ABB RAPID module: Código RAPID

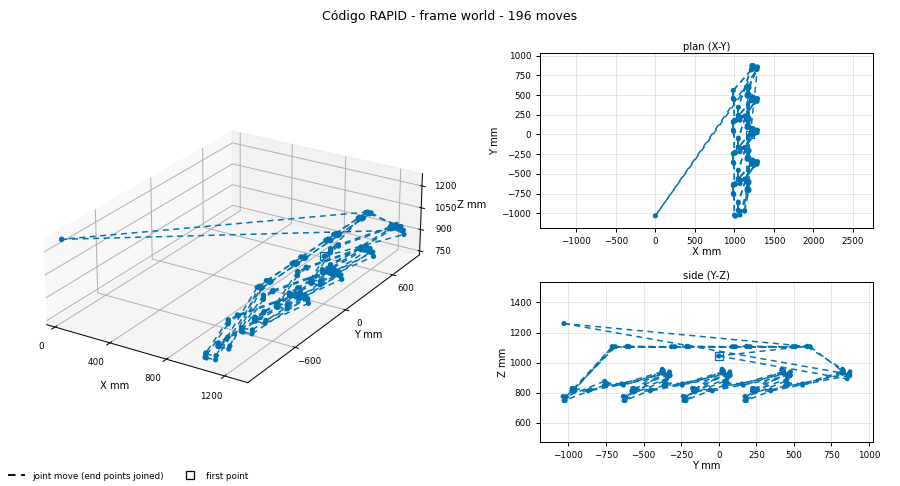
[picture p0: tool path of Código RAPID in frame world, 196 of 196 moves have a stored position in this frame; points joined in program order, loops and branches not executed]
MODULE Module1

    CONST robtarget HomeMesa:=[[1202.698927649,-0.006539298,1044.168012245],[0.707107406,0.00000178,0.707106156,-0.000001827],[-1,-1,0,1],[9E+09,9E+09,9E+09,0,0,0]];
    CONST robtarget Esperando:=[[0,-1030,1260],[0.500000347,0.500000347,0.499999653,-0.499999653],[-1,0,0,0],[9E+09,9E+09,9E+09,0,0,0]];
    CONST robtarget EsperandoMOVMesa:=[[-0.000045023,-1029.999947846,1260.000008248],[0.500000409,0.500000426,0.499999569,-0.499999596],[-2,0,0,0],[9E+09,9E+09,9E+09,180,0,0]];
    CONST robtarget HomeMesaDos:=[[1202.659544298,-0.000000047,1044.197481146],[0.706859937,0.00000059,0.707353539,0.00000059],[-1,-1,0,1],[9E+09,9E+09,9E+09,180,0,0]];
    CONST robtarget P1M1p1:=[[1294.65400628,854.62926339,891.446179617],[0.692157386,-0.14463472,0.692155179,-0.144638026],[0,0,-2,1],[9E+09,9E+09,9E+09,0,0,0]];
    CONST robtarget P1M1p2:=[[1240.529987934,870.337936268,911.143078471],[0.692157372,-0.144634704,0.692155207,-0.144637976],[0,0,-2,1],[9E+09,9E+09,9E+09,0,0,0]];
    CONST robtarget P1M1p3:=[[1227.787003999,873.332910408,915.014094682],[0.692157384,-0.144634674,0.692155202,-0.144637974],[0,0,-2,1],[9E+09,9E+09,9E+09,0,0,0]];
    CONST robtarget P1M1p4:=[[1222.239971547,870.997005167,915.013984808],[0.692157374,-0.144634683,0.692155208,-0.144637984],[0,0,-2,1],[9E+09,9E+09,9E+09,0,0,0]];
    CONST robtarget P1M1p5:=[[1050.485957284,345.048295942,811.300602855],[0.811802015,-0.047931337,0.525122518,0.250851384],[0,-1,0,1],[9E+09,9E+09,9E+09,0,0,0]];
    CONST robtarget P1M1p6:=[[1050.485947523,241.88479321,811.300594665],[0.811802009,-0.047931341,0.525122529,0.25085138],[0,-1,0,1],[9E+09,9E+09,9E+09,0,0,0]];
    CONST robtarget P1M1p7:=[[1057.883963041,232.826791757,811.30061261],[0.811802025,-0.047931351,0.525122498,0.250851392],[0,-1,0,1],[9E+09,9E+09,9E+09,0,0,0]];
    CONST robtarget P1M1p8:=[[1062.213995533,227.496594257,811.300605648],[0.81180201,-0.047931351,0.525122524,0.250851384],[0,-1,0,1],[9E+09,9E+09,9E+09,0,0,0]];
    CONST robtarget P1M1p9:=[[1069.026926797,223.929489315,811.300609594],[0.811802022,-0.047931351,0.525122506,0.250851385],[0,-1,0,1],[9E+09,9E+09,9E+09,0,0,0]];
    CONST robtarget P1M1p10:=[[1131.150947055,233.271896766,811.300583808],[0.811801999,-0.047931349,0.525122542,0.250851381],[0,-1,0,1],[9E+09,9E+09,9E+09,0,0,0]];
    CONST robtarget WaitMovMes1:=[[1202.698927649,-0.006539298,1044.168012245],[0.707107406,0.00000178,0.707106156,-0.000001827],[-1,-1,0,1],[9E+09,9E+09,9E+09,0,70,0]];
    CONST robtarget P1M1p11:=[[1185.930963599,608.173984403,1105.507035593],[0.707107406,0.000001819,0.707106156,-0.000001773],[0,0,-1,1],[9E+09,9E+09,9E+09,0,70,0]];
    CONST robtarget P1M1p12:=[[1185.930945833,510.993010056,1105.507039041],[0.707107406,0.000001805,0.707106157,-0.000001779],[0,0,-1,1],[9E+09,9E+09,9E+09,0,70,0]];
    CONST robtarget P1M2p1:=[[1287.081963914,823.391582063,930.460843736],[0.695385123,-0.126848673,0.695870584,-0.126937293],[0,0,-2,1],[9E+09,9E+09,9E+09,180,0,0]];
    CONST robtarget P1M2p2:=[[1232.892961405,829.555227251,930.460804282],[0.695385105,-0.126848727,0.69587059,-0.126937302],[0,0,-2,1],[9E+09,9E+09,9E+09,180,0,0]];
    CONST robtarget P1M2p3:=[[1217.609979435,827.253306759,930.460865831],[0.695385103,-0.12684871,0.695870597,-0.126937292],[0,0,-2,1],[9E+09,9E+09,9E+09,179.999964028,0,0]];
    CONST robtarget P1M2p4:=[[1214.009982986,817.991001642,930.460929766],[0.69538513,-0.126848699,0.695870573,-0.126937287],[0,0,-2,1],[9E+09,9E+09,9E+09,179.999964028,0,0]];
    CONST robtarget P1M2p5:=[[985.766137978,557.785104133,849.272525889],[0.8360719,0.017530565,0.547684306,0.026802208],[0,0,-1,1],[9E+09,9E+09,9E+09,179.999964028,0,0]];
    CONST robtarget P1M2p6:=[[985.766103061,457.716388895,849.272504479],[0.836071885,0.017530555,0.547684329,0.026802215],[0,0,-1,1],[9E+09,9E+09,9E+09,179.999964028,0,0]];
    CONST robtarget P1M2p7:=[[993.022666983,444.585787062,849.272520175],[0.836071898,0.017530568,0.547684309,0.026802211],[0,0,-1,1],[9E+09,9E+09,9E+09,179.999964028,0,0]];
    CONST robtarget P1M2p8:=[[1003.070938058,180.78768984,747.134418734],[0.807646496,0.209376596,0.514278881,0.19845859],[0,0,0,1],[9E+09,9E+09,9E+09,179.999964028,0,0]];
    CONST robtarget P1M2p9:=[[1013.977977246,173.442492628,747.1343984],[0.807646488,0.209376597,0.514278891,0.198458593],[0,0,0,1],[9E+09,9E+09,9E+09,179.999964028,0,0]];
    CONST robtarget P1M2p10:=[[1071.573952151,182.645606548,747.134407615],[0.807646513,0.209376602,0.514278845,0.198458605],[0,0,0,1],[9E+09,9E+09,9E+09,179.999964028,0,0]];
    CONST robtarget P1M2p11:=[[1185.930948842,588.452827755,1105.507011433],[0.707107409,0.000001805,0.707106154,-0.000001782],[0,0,-1,1],[9E+09,9E+09,9E+09,180,0,70]];
    CONST robtarget P1M2p12:=[[1185.93095036,492.129217368,1105.507026368],[0.707107404,0.000001839,0.707106158,-0.000001748],[0,0,-1,1],[9E+09,9E+09,9E+09,180,0,70]];
    CONST robtarget P2M1p1:=[[1294.653992166,454.43887346,891.446221022],[0.6921574,-0.144634673,0.692155181,-0.144638],[0,0,-1,1],[9E+09,9E+09,9E+09,0,0,0]];
    CONST robtarget P2M1p2:=[[1240.529984528,471.564123221,911.143162871],[0.692157397,-0.144634711,0.692155175,-0.144638006],[0,0,-1,1],[9E+09,9E+09,9E+09,0,0,0]];
    CONST robtarget P2M1p3:=[[1227.787003056,474.288594714,915.014113434],[0.69215739,-0.144634698,0.692155182,-0.144638018],[0,0,-1,1],[9E+09,9E+09,9E+09,0,0,0]];
    CONST robtarget P2M1p4:=[[1222.239953446,477.172888785,915.014065691],[0.692157397,-0.144634673,0.692155183,-0.144638],[0,0,-1,1],[9E+09,9E+09,9E+09,0,0,0]];
    CONST robtarget P2M1p5:=[[1050.485945509,-43.142440837,811.300594597],[0.811802019,-0.047931335,0.525122501,0.250851405],[-1,-1,0,1],[9E+09,9E+09,9E+09,0,0,0]];
    CONST robtarget P2M1p6:=[[1050.485952356,-156.521686759,811.300602341],[0.811802022,-0.047931365,0.525122503,0.250851385],[-1,-1,0,1],[9E+09,9E+09,9E+09,0,0,0]];
    CONST robtarget P2M1p7:=[[1057.883958265,-165.799494249,811.300583338],[0.811802006,-0.04793134,0.52512253,0.250851387],[-1,-1,0,1],[9E+09,9E+09,9E+09,0,0,0]];
    CONST robtarget P2M1p8:=[[1062.214006906,-168.868785565,811.300606455],[0.811802003,-0.047931336,0.525122535,0.250851386],[-1,-1,0,1],[9E+09,9E+09,9E+09,0,0,0]];
    CONST robtarget P2M1p9:=[[1069.026931582,-168.907600899,811.300592184],[0.811802005,-0.047931324,0.525122533,0.250851385],[-1,-1,0,1],[9E+09,9E+09,9E+09,0,0,0]];
    CONST robtarget P2M1p10:=[[1131.150939615,-165.021006485,811.300610263],[0.811802012,-0.047931365,0.525122515,0.250851394],[-1,-1,0,1],[9E+09,9E+09,9E+09,0,0,0]];
    CONST robtarget P2M1p11:=[[1185.930947732,209.275205026,1105.50703153],[0.707107405,0.00000183,0.707106157,-0.000001768],[0,0,-1,1],[9E+09,9E+09,9E+09,0,70,0]];
    CONST robtarget P2M1p12:=[[1185.930942037,104.027697243,1105.507044947],[0.707107412,0.000001825,0.70710615,-0.000001776],[0,0,-1,1],[9E+09,9E+09,9E+09,0,70,0]];
    CONST robtarget P3M1p1:=[[1294.653990055,54.307312118,891.446205655],[0.692157397,-0.144634698,0.692155177,-0.144638009],[0,0,-1,1],[9E+09,9E+09,9E+09,0,0,0]];
    CONST robtarget P3M1p2:=[[1240.529992729,70.522194984,911.143209882],[0.692157388,-0.144634701,0.692155185,-0.144638007],[0,0,-1,1],[9E+09,9E+09,9E+09,0,0,0]];
    CONST robtarget P3M1p3:=[[1227.787003035,75.815701326,915.01410237],[0.692157387,-0.144634691,0.692155191,-0.144637997],[0,0,-1,1],[9E+09,9E+09,9E+09,0,0,0]];
    CONST robtarget P3M1p4:=[[1222.239957402,75.077729076,915.014095799],[0.692157385,-0.144634702,0.692155189,-0.144638005],[0,0,-1,1],[9E+09,9E+09,9E+09,0,0,0]];
    CONST robtarget P3M1p5:=[[1050.485952963,-456.006186482,811.300606987],[0.811802017,-0.047931347,0.525122507,0.250851398],[-1,-1,0,1],[9E+09,9E+09,9E+09,0,0,0]];
    CONST robtarget P3M1p6:=[[1050.485949852,-556.041703529,811.300612034],[0.811802017,-0.047931384,0.525122509,0.250851386],[-1,-1,0,1],[9E+09,9E+09,9E+09,0,0,0]];
    CONST robtarget P3M1p7:=[[1057.883966107,-571.807786887,811.300587052],[0.811802004,-0.047931339,0.525122524,0.250851405],[-1,-1,0,1],[9E+09,9E+09,9E+09,0,0,0]];
    CONST robtarget P3M1p8:=[[1062.214003211,-570.695858455,811.30060674],[0.811802022,-0.047931361,0.525122502,0.25085139],[-1,-1,0,1],[9E+09,9E+09,9E+09,0,0,0]];
    CONST robtarget P3M1p9:=[[1069.02692125,-578.673501326,811.300606016],[0.811802025,-0.047931285,0.525122514,0.250851369],[-1,-1,0,1],[9E+09,9E+09,9E+09,0,0,0]];
    CONST robtarget P3M1p10:=[[1131.150956875,-570.701987213,811.300598508],[0.811802018,-0.047931365,0.525122499,0.250851406],[-1,-1,0,1],[9E+09,9E+09,9E+09,0,0,0]];
    CONST robtarget P3M1p11:=[[1185.930947007,-197.514283951,1105.507037733],[0.707107409,0.000001821,0.707106153,-0.00000177],[-1,-1,0,1],[9E+09,9E+09,9E+09,0,70,0]];
    CONST robtarget P3M1p12:=[[1185.930941597,-293.197607054,1105.507038781],[0.70710741,0.000001841,0.707106152,-0.000001751],[-1,-1,0,1],[9E+09,9E+09,9E+09,0,70,0]];
    CONST robtarget P4M1p1:=[[1294.653989986,-345.662907333,891.446190924],[0.692157389,-0.144634676,0.69215519,-0.144638004],[-1,-1,0,1],[9E+09,9E+09,9E+09,0,0,0]];
    CONST robtarget P4M1p2:=[[1240.530000685,-329.603196599,911.143191009],[0.692157385,-0.1446347,0.692155189,-0.144638003],[-1,-1,0,1],[9E+09,9E+09,9E+09,0,0,0]];
    CONST robtarget P4M1p3:=[[1227.787004205,-322.940201758,915.014096584],[0.692157384,-0.144634687,0.692155193,-0.144638003],[-1,-1,0,1],[9E+09,9E+09,9E+09,0,0,0]];
    CONST robtarget P4M1p4:=[[1222.23995583,-327.607308393,915.014097519],[0.692157385,-0.144634701,0.692155189,-0.144638006],[-1,-1,0,1],[9E+09,9E+09,9E+09,0,0,0]];
    CONST robtarget P4M1p5:=[[1050.485949411,-869.115712575,811.300612218],[0.811802019,-0.047931325,0.525122516,0.250851378],[-1,-1,0,1],[9E+09,9E+09,9E+09,0,0,0]];
    CONST robtarget P4M1p6:=[[1050.485974835,-958.232069962,811.300585733],[0.811802011,-0.047931384,0.525122503,0.250851418],[-1,-1,0,1],[9E+09,9E+09,9E+09,0,0,0]];
    CONST robtarget P4M1p7:=[[1057.88399001,-975.404649155,811.30060734],[0.811802006,-0.047931318,0.525122528,0.250851396],[-1,-1,0,1],[9E+09,9E+09,9E+09,0,0,0]];
    CONST robtarget P4M1p8:=[[1062.214034381,-973.918880257,811.300571248],[0.811802021,-0.047931344,0.525122509,0.250851381],[-1,-1,0,1],[9E+09,9E+09,9E+09,0,0,0]];
    CONST robtarget P4M1p9:=[[1069.026916149,-978.501930546,811.300562057],[0.811802023,-0.047931276,0.525122506,0.250851395],[-1,-1,0,1],[9E+09,9E+09,9E+09,0,0,0]];
    CONST robtarget P4M1p10:=[[1131.150931317,-972.859035446,811.300552906],[0.811802013,-0.047931366,0.525122516,0.250851386],[-1,-1,0,1],[9E+09,9E+09,9E+09,0,0,0]];
    CONST robtarget P4M1p11:=[[1185.930958357,-596.032669183,1105.507027322],[0.70710741,0.000001831,0.707106152,-0.000001743],[-1,-1,0,1],[9E+09,9E+09,9E+09,0,70,0]];
    CONST robtarget P4M1p12:=[[1185.930974143,-694.807857486,1105.507021321],[0.707107404,0.000001822,0.707106159,-0.000001766],[-1,-1,0,1],[9E+09,9E+09,9E+09,0,70,0]];
    CONST robtarget TurnMesa:=[[1202.698927649,-0.006539298,1044.168012245],[0.707107406,0.00000178,0.707106156,-0.000001827],[-1,-1,0,1],[9E+09,9E+09,9E+09,0,180,0]];
    CONST robtarget P5M1p1:=[[1287.51280176,856.97594778,918.184846829],[0.692157388,-0.144634706,0.692155182,-0.144638018],[0,0,-2,1],[9E+09,9E+09,9E+09,0,180,0]];
    CONST robtarget P5M1p2:=[[1240.529986137,870.338041259,927.422439494],[0.69215738,-0.144634719,0.692155189,-0.144638011],[0,0,-2,1],[9E+09,9E+09,9E+09,0,180,0]];
    CONST robtarget P5M1p3:=[[1227.787003999,873.332910408,938.961164099],[0.692157384,-0.144634674,0.692155202,-0.144637974],[0,0,-2,1],[9E+09,9E+09,9E+09,0,180,0]];
    CONST robtarget P5M1p4:=[[1222.239971547,870.997005167,929.420285517],[0.692157374,-0.144634683,0.692155208,-0.144637984],[0,0,-2,1],[9E+09,9E+09,9E+09,0,180,0]];
    CONST robtarget P5M1p5:=[[1050.485957284,345.048295942,818.663201985],[0.811802015,-0.047931337,0.525122518,0.250851384],[0,-1,0,1],[9E+09,9E+09,9E+09,0,180,0]];
    CONST robtarget P5M1p6:=[[1050.485947523,241.88479321,824.353888262],[0.811802009,-0.047931341,0.525122529,0.25085138],[0,-1,0,1],[9E+09,9E+09,9E+09,0,180,0]];
    CONST robtarget P5M1p7:=[[1057.883963041,232.826791757,825.451999614],[0.811802025,-0.047931351,0.525122498,0.250851392],[0,-1,0,1],[9E+09,9E+09,9E+09,0,180,0]];
    CONST robtarget P5M1p8:=[[1062.213995533,227.496594257,827.795822741],[0.81180201,-0.047931351,0.525122524,0.250851384],[0,-1,0,1],[9E+09,9E+09,9E+09,0,180,0]];
    CONST robtarget P5M1p9:=[[1069.026926797,223.929489315,828.586291332],[0.811802022,-0.047931351,0.525122506,0.250851385],[0,-1,0,1],[9E+09,9E+09,9E+09,0,180,0]];
    CONST robtarget P5M1p10:=[[1131.150947055,233.271896766,826.446924128],[0.811801999,-0.047931349,0.525122542,0.250851381],[0,-1,0,1],[9E+09,9E+09,9E+09,0,180,0]];
    CONST robtarget P5M1p11:=[[1160.941867257,608.173984403,1105.507035593],[0.707107406,0.000001819,0.707106156,-0.000001773],[0,0,-1,1],[9E+09,9E+09,9E+09,0,250,0]];
    CONST robtarget P5M1p12:=[[1160.941943935,507.930686372,1105.50702957],[0.707107404,0.000001805,0.707106158,-0.000001799],[0,0,-1,1],[9E+09,9E+09,9E+09,0,250,0]];
    CONST robtarget P6M1p1:=[[1287.512992537,455.226798507,918.184930623],[0.692157396,-0.14463471,0.692155172,-0.144638022],[0,0,-1,1],[9E+09,9E+09,9E+09,0,180,0]];
    CONST robtarget P6M1p2:=[[1240.530007914,466.532478263,927.422537461],[0.692157392,-0.14463468,0.692155189,-0.144637993],[0,0,-1,1],[9E+09,9E+09,9E+09,0,180,0]];
    CONST robtarget P6M1p3:=[[1227.787004184,477.674601054,938.961099959],[0.692157386,-0.144634703,0.692155187,-0.14463801],[0,0,-1,1],[9E+09,9E+09,9E+09,0,180,0]];
    CONST robtarget P6M1p4:=[[1222.239961288,469.693192082,929.420433939],[0.69215739,-0.144634696,0.692155187,-0.144637993],[0,0,-1,1],[9E+09,9E+09,9E+09,0,180,0]];
    CONST robtarget P6M1p5:=[[1050.485946451,-57.179143328,818.663195557],[0.81180201,-0.04793132,0.525122533,0.250851372],[-1,-1,0,1],[9E+09,9E+09,9E+09,0,180,0]];
    CONST robtarget P6M1p6:=[[1050.485945699,-158.82959493,824.353885396],[0.811802018,-0.047931342,0.525122505,0.250851399],[-1,-1,0,1],[9E+09,9E+09,9E+09,0,180,0]];
    CONST robtarget P6M1p7:=[[1057.883963528,-170.135898305,825.452052847],[0.811802002,-0.047931347,0.525122534,0.250851389],[-1,-1,0,1],[9E+09,9E+09,9E+09,0,180,0]];
    CONST robtarget P6M1p8:=[[1062.213999596,-173.347293692,827.795942722],[0.811802007,-0.047931318,0.525122528,0.250851393],[-1,-1,0,1],[9E+09,9E+09,9E+09,0,180,0]];
    CONST robtarget P6M1p9:=[[1069.02693064,-173.705298015,828.586300968],[0.811802009,-0.047931353,0.525122532,0.250851372],[-1,-1,0,1],[9E+09,9E+09,9E+09,0,180,0]];
    CONST robtarget P6M1p10:=[[1131.15094581,-164.207103159,826.447012387],[0.811802001,-0.047931347,0.525122543,0.250851374],[-1,-1,0,1],[9E+09,9E+09,9E+09,0,180,0]];
    CONST robtarget P7M1p1:=[[1287.5130039,55.947838621,918.184889325],[0.69215739,-0.1446347,0.692155182,-0.14463801],[0,0,-1,1],[9E+09,9E+09,9E+09,0,180,0]];
    CONST robtarget P7M1p2:=[[1240.529993957,74.049824175,927.422605126],[0.692157388,-0.144634689,0.69215519,-0.144637995],[0,0,-1,1],[9E+09,9E+09,9E+09,0,180,0]];
    CONST robtarget P7M1p3:=[[1227.786997792,73.453377394,938.961112671],[0.692157392,-0.144634702,0.69215518,-0.144638014],[0,0,-1,1],[9E+09,9E+09,9E+09,0,180,0]];
    CONST robtarget P7M1p4:=[[1222.239945235,71.066640414,929.420450662],[0.692157398,-0.144634691,0.692155178,-0.144638003],[0,0,-1,1],[9E+09,9E+09,9E+09,0,180,0]];
    CONST robtarget P7M1p5:=[[1050.485943723,-450.547007586,818.663211154],[0.811802031,-0.047931305,0.525122495,0.250851388],[-1,-1,0,1],[9E+09,9E+09,9E+09,0,180,0]];
    CONST robtarget P7M1p6:=[[1050.485951308,-555.654089777,824.353906332],[0.811802023,-0.047931345,0.525122502,0.25085139],[-1,-1,0,1],[9E+09,9E+09,9E+09,0,180,0]];
    CONST robtarget P7M1p7:=[[1057.883971379,-565.529692139,825.452046896],[0.811802007,-0.047931352,0.525122531,0.250851378],[-1,-1,0,1],[9E+09,9E+09,9E+09,0,180,0]];
    CONST robtarget P7M1p8:=[[1062.214013779,-572.186553681,827.795959878],[0.811802015,-0.047931347,0.525122524,0.250851369],[-1,-1,0,1],[9E+09,9E+09,9E+09,0,180,0]];
    CONST robtarget P7M1p9:=[[1069.026937537,-571.189267924,828.58630883],[0.811802019,-0.047931339,0.525122522,0.250851362],[-1,-1,0,1],[9E+09,9E+09,9E+09,0,180,0]];
    CONST robtarget P7M1p10:=[[1131.150959132,-562.660960026,826.447030815],[0.81180201,-0.047931389,0.525122518,0.25085139],[-1,-1,0,1],[9E+09,9E+09,9E+09,0,180,0]];
    CONST robtarget P6M1p11:=[[1160.941935741,207.369302139,1105.50703556],[0.707107406,0.000001794,0.707106157,-0.00000179],[0,0,-1,1],[9E+09,9E+09,9E+09,0,250,0]];
    CONST robtarget P6M1p12:=[[1160.941940446,113.055695188,1105.507031057],[0.707107406,0.00000181,0.707106156,-0.000001778],[0,0,-1,1],[9E+09,9E+09,9E+09,0,250,0]];
    CONST robtarget P7M1p11:=[[1160.941939753,-202.48499324,1105.507031431],[0.707107406,0.00000177,0.707106157,-0.000001802],[-1,-1,0,1],[9E+09,9E+09,9E+09,0,250,0]];
    CONST robtarget P7M1p12:=[[1160.941939671,-291.239289206,1105.507030754],[0.70710741,0.000001779,0.707106153,-0.000001789],[-1,-1,0,1],[9E+09,9E+09,9E+09,0,250,0]];
    CONST robtarget P8M1p1:=[[1287.513001746,-341.869412046,918.184887932],[0.692157384,-0.144634701,0.69215519,-0.144638003],[-1,-1,0,1],[9E+09,9E+09,9E+09,0,180,0]];
    CONST robtarget P8M1p2:=[[1240.529989369,-331.61750501,927.422616777],[0.692157392,-0.144634697,0.692155182,-0.144638007],[-1,-1,0,1],[9E+09,9E+09,9E+09,0,180,0]];
    CONST robtarget P8M1p3:=[[1227.787006733,-328.052388339,938.961097781],[0.692157382,-0.144634706,0.692155192,-0.144638003],[-1,-1,0,1],[9E+09,9E+09,9E+09,0,180,0]];
    CONST robtarget P8M1p4:=[[1222.23995944,-330.109669308,929.420486052],[0.692157392,-0.144634689,0.692155187,-0.144637993],[-1,-1,0,1],[9E+09,9E+09,9E+09,0,180,0]];
    CONST robtarget P8M1p5:=[[1050.485978825,-853.276272126,818.663203151],[0.81180201,-0.047931328,0.525122523,0.250851391],[-1,-1,0,1],[9E+09,9E+09,9E+09,0,180,0]];
    CONST robtarget P8M1p6:=[[1050.485957025,-958.593434584,824.353874621],[0.811802012,-0.047931339,0.525122527,0.250851375],[-1,-1,0,1],[9E+09,9E+09,9E+09,0,180,0]];
    CONST robtarget P8M1p7:=[[1057.883978797,-972.736439335,825.452068596],[0.811802005,-0.047931352,0.525122524,0.250851402],[-1,-1,0,1],[9E+09,9E+09,9E+09,0,180,0]];
    CONST robtarget P8M1p8:=[[1062.214032655,-971.575289729,827.795997264],[0.811802013,-0.047931351,0.525122523,0.250851377],[-1,-1,0,1],[9E+09,9E+09,9E+09,0,180,0]];
    CONST robtarget P8M1p9:=[[1069.026937278,-976.446817795,828.586268385],[0.811802017,-0.047931332,0.525122513,0.250851388],[-1,-1,0,1],[9E+09,9E+09,9E+09,0,180,0]];
    CONST robtarget P8M1p10:=[[1131.150976145,-960.905988949,826.447126012],[0.811802005,-0.047931424,0.525122525,0.250851386],[-1,-1,0,1],[9E+09,9E+09,9E+09,0,180,0]];
    CONST robtarget P8M1p11:=[[1160.941952888,-598.731774088,1105.507053568],[0.707107405,0.000001738,0.707106157,-0.000001833],[-1,-1,0,1],[9E+09,9E+09,9E+09,0,250,0]];
    CONST robtarget P8M1p12:=[[1160.941938987,-686.786158028,1105.507050864],[0.70710742,0.00000173,0.707106142,-0.00000184],[-1,-1,0,1],[9E+09,9E+09,9E+09,0,250,0]];
    CONST robtarget P2M2p1:=[[1287.081942915,423.299490757,930.460887717],[0.695385109,-0.1268487,0.695870591,-0.126937301],[0,0,-1,1],[9E+09,9E+09,9E+09,180,0,0]];
    CONST robtarget P2M2p2:=[[1232.892982774,430.194982931,930.460817958],[0.695385103,-0.126848709,0.695870593,-0.126937314],[0,0,-1,1],[9E+09,9E+09,9E+09,180,0,0]];
    CONST robtarget P2M2p3:=[[1217.609985933,434.601968819,930.460907436],[0.695385116,-0.126848706,0.69587058,-0.126937316],[0,0,-1,1],[9E+09,9E+09,9E+09,180,0,0]];
    CONST robtarget P2M2p4:=[[1214.009978094,428.335193568,930.460893887],[0.695385201,-0.126848703,0.6958705,-0.126937292],[0,0,-1,1],[9E+09,9E+09,9E+09,180,0,0]];
    CONST robtarget P2M2p5:=[[985.766084152,163.956301034,849.272497669],[0.836071892,0.017530565,0.547684317,0.02680222],[0,0,-1,1],[9E+09,9E+09,9E+09,180,0,0]];
    CONST robtarget P2M2p6:=[[985.7660988,48.871628128,849.272538428],[0.836071912,0.01753054,0.547684287,0.02680222],[0,0,0,1],[9E+09,9E+09,9E+09,180,0,0]];
    CONST robtarget P2M2p7:=[[993.022664863,36.972499936,849.272528775],[0.8360719,0.017530569,0.547684306,0.02680221],[0,0,0,1],[9E+09,9E+09,9E+09,180,0,0]];
    CONST robtarget P2M2p8:=[[1003.0709257,-228.723692996,747.134400051],[0.807646484,0.209376611,0.514278887,0.198458605],[-1,-1,0,1],[9E+09,9E+09,9E+09,180,0,0]];
    CONST robtarget P2M2p9:=[[1013.977992175,-232.129697703,747.134426921],[0.807646515,0.209376583,0.514278857,0.198458586],[-1,-1,0,1],[9E+09,9E+09,9E+09,180,0,0]];
    CONST robtarget P2M2p10:=[[1071.573958877,-217.594289105,747.13441737],[0.80764653,0.209376599,0.514278819,0.198458606],[-1,-1,0,1],[9E+09,9E+09,9E+09,180,0,0]];
    CONST robtarget P2M2p11:=[[1185.930950239,187.675889547,1105.507032353],[0.707107407,0.000001823,0.707106155,-0.000001789],[0,0,-1,1],[9E+09,9E+09,9E+09,180,0,70]];
    CONST robtarget P2M2p12:=[[1185.930943233,95.529018748,1105.507041573],[0.70710741,0.000001834,0.707106153,-0.000001752],[0,0,-1,1],[9E+09,9E+09,9E+09,180,0,70]];
    CONST robtarget P3M2p1:=[[1287.081941566,21.413279151,930.460887197],[0.695385111,-0.126848701,0.695870588,-0.126937304],[0,0,-1,1],[9E+09,9E+09,9E+09,180,0,0]];
    CONST robtarget P3M2p2:=[[1232.892967953,28.987158369,930.460840817],[0.695385113,-0.126848699,0.695870587,-0.126937303],[0,0,-1,1],[9E+09,9E+09,9E+09,180,0,0]];
    CONST robtarget P3M2p3:=[[1217.60998262,34.410408763,930.460892089],[0.695385108,-0.126848696,0.695870593,-0.126937298],[0,0,-1,1],[9E+09,9E+09,9E+09,180,0,0]];
    CONST robtarget P3M2p4:=[[1214.009984068,31.687269665,930.460885715],[0.695385201,-0.126848699,0.695870499,-0.126937302],[0,0,-1,1],[9E+09,9E+09,9E+09,180,0,0]];
    CONST robtarget P3M2p5:=[[985.766085968,-242.896799387,849.27250766],[0.836071903,0.017530563,0.547684302,0.026802208],[-1,-1,0,1],[9E+09,9E+09,9E+09,180,0,0]];
    CONST robtarget P3M2p6:=[[985.766092573,-352.969410753,849.272514142],[0.836071905,0.017530541,0.547684299,0.026802214],[-1,-1,0,1],[9E+09,9E+09,9E+09,180,0,0]];
    CONST robtarget P3M2p7:=[[993.022662409,-364.919381115,849.272509954],[0.83607191,0.017530563,0.547684291,0.026802221],[-1,-1,0,1],[9E+09,9E+09,9E+09,180,0,0]];
    CONST robtarget P3M2p8:=[[1003.070932407,-628.513700129,747.134415648],[0.807646507,0.209376596,0.51427886,0.198458599],[-1,-1,0,1],[9E+09,9E+09,9E+09,180,0,0]];
    CONST robtarget P3M2p9:=[[1013.977996648,-630.345557467,747.134426277],[0.807646526,0.209376596,0.514278831,0.198458594],[-1,-1,0,1],[9E+09,9E+09,9E+09,180,0,0]];
    CONST robtarget P3M2p10:=[[1071.573965127,-622.825071858,747.134417066],[0.807646527,0.209376586,0.514278841,0.198458579],[-1,-1,0,1],[9E+09,9E+09,9E+09,180,0,0]];
    CONST robtarget P3M2p11:=[[1185.930946533,-213.064594931,1105.507036914],[0.707107409,0.000001806,0.707106153,-0.000001799],[-1,-1,0,1],[9E+09,9E+09,9E+09,180,0,70]];
    CONST robtarget P3M2p12:=[[1185.930948227,-314.722485056,1105.507040307],[0.707107408,0.0000018,0.707106154,-0.000001796],[-1,-1,0,1],[9E+09,9E+09,9E+09,180,0,70]];
    CONST robtarget P4M2p1:=[[1287.081937875,-376.65299891,930.46088109],[0.695385101,-0.126848707,0.695870596,-0.126937313],[-1,-1,0,1],[9E+09,9E+09,9E+09,180,0,0]];
    CONST robtarget P4M2p2:=[[1232.892982402,-370.043883982,930.460878188],[0.695385103,-0.126848708,0.695870596,-0.126937299],[-1,-1,0,1],[9E+09,9E+09,9E+09,180,0,0]];
    CONST robtarget P4M2p3:=[[1217.609984921,-367.718324415,930.460875748],[0.695385104,-0.126848682,0.695870599,-0.126937299],[-1,-1,0,1],[9E+09,9E+09,9E+09,180,0,0]];
    CONST robtarget P4M2p4:=[[1214.009976161,-372.318596656,930.460900471],[0.695385203,-0.126848704,0.695870495,-0.126937304],[-1,-1,0,1],[9E+09,9E+09,9E+09,180,0,0]];
    CONST robtarget P4M2p5:=[[985.766087685,-634.35829981,849.272500138],[0.836071901,0.017530576,0.547684304,0.02680221],[-1,-1,0,1],[9E+09,9E+09,9E+09,180,0,0]];
    CONST robtarget P4M2p6:=[[985.766074892,-747.923087794,849.272525035],[0.836071911,0.017530544,0.54768429,0.026802203],[-1,-1,0,1],[9E+09,9E+09,9E+09,180,0,0]];
    CONST robtarget P4M2p7:=[[993.022657334,-761.317316304,849.272520024],[0.836071894,0.017530573,0.547684315,0.026802205],[-1,-1,0,1],[9E+09,9E+09,9E+09,180,0,0]];
    CONST robtarget P4M2p8:=[[1003.070923563,-1027.52495413,747.134373101],[0.807646499,0.209376593,0.514278873,0.198458599],[-1,-1,0,1],[9E+09,9E+09,9E+09,180,0,0]];
    CONST robtarget P4M2p9:=[[1013.978011173,-1030.027003938,747.13443015],[0.807646524,0.209376598,0.514278843,0.19845857],[-1,-1,0,1],[9E+09,9E+09,9E+09,180,0,0]];
    CONST robtarget P4M2p10:=[[1071.573975734,-1021.038991656,747.134380172],[0.807646517,0.209376617,0.514278826,0.198458622],[-1,-1,0,1],[9E+09,9E+09,9E+09,180,0,0]];
    CONST robtarget P4M2p11:=[[1185.930951631,-611.718126779,1105.50700953],[0.707107393,0.000001797,0.707106169,-0.000001819],[-1,-1,0,1],[9E+09,9E+09,9E+09,180,0,70]];
    CONST robtarget P4M2p12:=[[1185.930932946,-710.183230163,1105.507022383],[0.707107409,0.000001848,0.707106153,-0.000001799],[-1,-1,0,1],[9E+09,9E+09,9E+09,180,0,70]];
    CONST robtarget P5M2p1:=[[1287.081963937,823.39158063,956.573530849],[0.695385109,-0.126848705,0.695870584,-0.126937335],[0,0,-2,1],[9E+09,9E+09,9E+09,180,0,180]];
    CONST robtarget P5M2p2:=[[1232.892961405,829.555227251,946.574452649],[0.695385105,-0.126848727,0.69587059,-0.126937302],[0,0,-2,1],[9E+09,9E+09,9E+09,180,0,180]];
    CONST robtarget P5M2p3:=[[1217.609979435,827.253306759,946.518852379],[0.695385103,-0.12684871,0.695870597,-0.126937292],[0,0,-2,1],[9E+09,9E+09,9E+09,180,0,180]];
    CONST robtarget P5M2p4:=[[1214.009981629,817.991000196,938.720837099],[0.695385178,-0.126848677,0.695870529,-0.126937286],[0,0,-2,1],[9E+09,9E+09,9E+09,180,0,180]];
    CONST robtarget P5M2p5:=[[985.766096585,557.785078701,859.297655027],[0.836071893,0.017530567,0.547684317,0.026802216],[0,0,-1,1],[9E+09,9E+09,9E+09,180,0,180]];
    CONST robtarget P5M2p6:=[[985.766102672,457.71639088,863.722348668],[0.836071888,0.017530541,0.547684325,0.026802215],[0,0,-1,1],[9E+09,9E+09,9E+09,180,0,180]];
    CONST robtarget P5M2p7:=[[993.022666983,444.585787062,876.038087888],[0.836071898,0.017530568,0.547684309,0.026802211],[0,0,-1,1],[9E+09,9E+09,9E+09,180,0,180]];
    CONST robtarget P5M2p8:=[[1003.070938058,180.78768984,772.485475081],[0.807646496,0.209376596,0.514278881,0.19845859],[0,0,0,1],[9E+09,9E+09,9E+09,180,0,180]];
    CONST robtarget P5M2p9:=[[1013.977977246,173.442492628,774.873565047],[0.807646488,0.209376597,0.514278891,0.198458593],[0,0,0,1],[9E+09,9E+09,9E+09,180,0,180]];
    CONST robtarget P5M2p10:=[[1071.573952151,182.645606548,771.890741042],[0.807646513,0.209376602,0.514278845,0.198458605],[0,0,0,1],[9E+09,9E+09,9E+09,180,0,180]];
    CONST robtarget P5M2p11:=[[1159.718533142,588.452792411,1109.600135223],[0.707107409,0.000001816,0.707106154,-0.000001793],[0,0,-1,1],[9E+09,9E+09,9E+09,180,0,250]];
    CONST robtarget P5M2p12:=[[1158.995416353,492.129217368,1105.507026368],[0.707107404,0.000001839,0.707106158,-0.000001748],[0,0,-1,1],[9E+09,9E+09,9E+09,180,0,250]];
    CONST robtarget P6M2p1:=[[1287.081942874,420.03000634,956.573432269],[0.69538511,-0.126848716,0.695870585,-0.126937314],[0,0,-1,1],[9E+09,9E+09,9E+09,180,0,180]];
    CONST robtarget P6M2p2:=[[1232.892962329,427.246392285,946.574422328],[0.695385114,-0.126848699,0.695870586,-0.1269373],[0,0,-1,1],[9E+09,9E+09,9E+09,180,0,180]];
    CONST robtarget P6M2p3:=[[1217.609978669,431.701906072,946.518805799],[0.695385111,-0.126848707,0.695870589,-0.126937293],[0,0,-1,1],[9E+09,9E+09,9E+09,180,0,180]];
    CONST robtarget P6M2p4:=[[1214.009982742,425.527880519,938.720915064],[0.695385203,-0.12684869,0.6958705,-0.126937297],[0,0,-1,1],[9E+09,9E+09,9E+09,180,0,180]];
    CONST robtarget P6M2p5:=[[985.766086342,153.560690225,859.297582324],[0.836071893,0.01753055,0.547684317,0.026802227],[0,0,-1,1],[9E+09,9E+09,9E+09,180,0,180]];
    CONST robtarget P6M2p6:=[[985.766094733,57.430100166,863.7224247],[0.83607191,0.01753054,0.54768429,0.026802231],[0,0,-1,1],[9E+09,9E+09,9E+09,180,0,180]];
    CONST robtarget P6M2p7:=[[993.022659885,38.244880974,876.038102784],[0.836071901,0.01753056,0.547684304,0.02680221],[0,0,0,1],[9E+09,9E+09,9E+09,180,0,180]];
    CONST robtarget P6M2p8:=[[1003.070925748,-229.263088707,772.48562708],[0.807646486,0.20937661,0.514278885,0.198458604],[-1,-1,0,1],[9E+09,9E+09,9E+09,180,0,180]];
    CONST robtarget P6M2p9:=[[1013.977986109,-237.325696282,774.87363237],[0.807646493,0.209376602,0.514278882,0.19845859],[-1,-1,0,1],[9E+09,9E+09,9E+09,180,0,180]];
    CONST robtarget P6M2p10:=[[1071.5739537,-217.291392288,771.890844811],[0.807646529,0.209376602,0.514278817,0.198458612],[-1,-1,0,1],[9E+09,9E+09,9E+09,180,0,180]];
    CONST robtarget P6M2p11:=[[1159.718967768,185.056293345,1109.599968508],[0.707107406,0.000001782,0.707106157,-0.000001809],[0,0,-1,1],[9E+09,9E+09,9E+09,180,0,250]];
    CONST robtarget P6M2p12:=[[1158.995007718,88.334741652,1105.507040855],[0.707107407,0.000001845,0.707106155,-0.000001754],[0,0,-1,1],[9E+09,9E+09,9E+09,180,0,250]];
    CONST robtarget P7M2p1:=[[1287.081938268,21.890938974,956.57351039],[0.695385113,-0.126848703,0.695870585,-0.126937308],[0,0,-1,1],[9E+09,9E+09,9E+09,180,0,180]];
    CONST robtarget P7M2p2:=[[1232.89296877,24.144487835,946.574415906],[0.695385111,-0.126848702,0.695870587,-0.126937306],[0,0,-1,1],[9E+09,9E+09,9E+09,180,0,180]];
    CONST robtarget P7M2p3:=[[1217.609978031,30.830878938,946.518813687],[0.695385117,-0.126848694,0.695870584,-0.126937301],[0,0,-1,1],[9E+09,9E+09,9E+09,180,0,180]];
    CONST robtarget P7M2p4:=[[1214.009982564,27.014900378,938.720897759],[0.695385201,-0.126848692,0.695870501,-0.126937294],[0,0,-1,1],[9E+09,9E+09,9E+09,180,0,180]];
    CONST robtarget P7M2p5:=[[985.766097151,-242.694294826,859.297602362],[0.836071894,0.017530542,0.547684315,0.026802225],[-1,-1,0,1],[9E+09,9E+09,9E+09,180,0,180]];
    CONST robtarget P7M2p6:=[[985.766099125,-352.829883584,863.722418914],[0.836071911,0.017530532,0.547684288,0.026802244],[-1,-1,0,1],[9E+09,9E+09,9E+09,180,0,180]];
    CONST robtarget P7M2p7:=[[993.022660819,-362.965703245,876.038079243],[0.836071881,0.017530584,0.547684334,0.026802208],[-1,-1,0,1],[9E+09,9E+09,9E+09,180,0,180]];
    CONST robtarget P7M2p8:=[[1003.070948251,-628.753993071,772.485658081],[0.807646515,0.209376563,0.514278862,0.198458594],[-1,-1,0,1],[9E+09,9E+09,9E+09,180,0,180]];
    CONST robtarget P7M2p9:=[[1013.977972406,-636.678405216,774.873711553],[0.807646507,0.209376587,0.514278867,0.19845859],[-1,-1,0,1],[9E+09,9E+09,9E+09,180,0,180]];
    CONST robtarget P7M2p10:=[[1071.573961903,-618.428809445,771.890835972],[0.80764652,0.209376611,0.514278821,0.198458631],[-1,-1,0,1],[9E+09,9E+09,9E+09,180,0,180]];
    CONST robtarget P7M2p11:=[[1159.718972896,-211.532582055,1109.599963477],[0.707107406,0.000001788,0.707106156,-0.000001804],[-1,-1,0,1],[9E+09,9E+09,9E+09,180,0,250]];
    CONST robtarget P7M2p12:=[[1158.995014498,-312.213370951,1105.507037983],[0.707107405,0.000001806,0.707106158,-0.000001779],[-1,-1,0,1],[9E+09,9E+09,9E+09,180,0,250]];
    CONST robtarget P8M2p1:=[[1287.081946207,-375.923966976,956.573509614],[0.695385119,-0.126848699,0.695870583,-0.126937291],[-1,-1,0,1],[9E+09,9E+09,9E+09,180,0,180]];
    CONST robtarget P8M2p2:=[[1232.892963196,-371.870194113,946.57442583],[0.69538511,-0.1268487,0.695870588,-0.126937308],[-1,-1,0,1],[9E+09,9E+09,9E+09,180,0,180]];
    CONST robtarget P8M2p3:=[[1217.609976063,-368.396995577,946.518812071],[0.695385112,-0.126848691,0.695870589,-0.126937305],[-1,-1,0,1],[9E+09,9E+09,9E+09,180,0,180]];
    CONST robtarget P8M2p4:=[[1214.009980014,-377.44629786,938.720900615],[0.695385192,-0.126848698,0.695870507,-0.126937304],[-1,-1,0,1],[9E+09,9E+09,9E+09,180,0,180]];
    CONST robtarget P8M2p5:=[[985.766102139,-645.865947475,859.297609634],[0.83607191,0.017530516,0.54768429,0.026802252],[-1,-1,0,1],[9E+09,9E+09,9E+09,180,0,180]];
    CONST robtarget P8M2p6:=[[985.766111508,-745.745453353,863.722406721],[0.836071896,0.017530535,0.547684312,0.026802244],[-1,-1,0,1],[9E+09,9E+09,9E+09,180,0,180]];
    CONST robtarget P8M2p7:=[[993.022651473,-759.598032516,876.03808882],[0.836071897,0.017530614,0.547684309,0.026802201],[-1,-1,0,1],[9E+09,9E+09,9E+09,180,0,180]];
    CONST robtarget P8M2p8:=[[1003.070942622,-1018.707021048,772.485722249],[0.807646501,0.209376576,0.514278888,0.198458571],[-1,-1,0,1],[9E+09,9E+09,9E+09,180,0,180]];
    CONST robtarget P8M2p9:=[[1013.978003834,-1036.740997077,774.873673039],[0.8076465,0.209376594,0.514278873,0.198458597],[-1,-1,0,1],[9E+09,9E+09,9E+09,180,0,180]];
    CONST robtarget P8M2p10:=[[1071.573951587,-1017.140980769,771.890848396],[0.807646521,0.209376617,0.514278833,0.19845859],[-1,-1,0,1],[9E+09,9E+09,9E+09,180,0,180]];
    CONST robtarget P8M2p11:=[[1159.718972934,-607.249324049,1109.599962504],[0.707107405,0.000001767,0.707106157,-0.00000183],[-1,-1,0,1],[9E+09,9E+09,9E+09,180,0,250]];
    CONST robtarget P8M2p12:=[[1158.994998413,-707.410705769,1105.507042887],[0.707107419,0.000001829,0.707106143,-0.000001755],[-1,-1,0,1],[9E+09,9E+09,9E+09,180,0,250]];
!***********************************************************
    !
    ! Module:  Module1
    !
    ! Description:
    !   <Insert description here>
    !
    ! Author: robertoruiz
    !
    ! Version: 1.0
    !
    !***********************************************************


    !***********************************************************
    !
    ! Procedure main
    !
    !   This is the entry point of your program
    !
    !***********************************************************
    PROC main()
        !Add your code here
        ActUnit INTERCH;
        MoveJ HomeMesa,v1000,z100,tool0\WObj:=wobj0;
        MoveJ P1M1p1,v1000,z100,tool0\WObj:=wobj0;
        MoveJ P1M1p2,v40,z100,tool0\WObj:=wobj0;
        MoveJ P1M1p3,v40,z100,tool0\WObj:=wobj0;
        MoveJ P1M1p4,v40,z100,tool0\WObj:=wobj0;
        MoveJ P1M1p5,v1500,z100,tool0\WObj:=wobj0;
        MoveJ P1M1p6,v40,z100,tool0\WObj:=wobj0;
        MoveJ P1M1p7,v1500,z100,tool0\WObj:=wobj0;
        MoveJ P1M1p8,v40,z100,tool0\WObj:=wobj0;
        MoveJ P1M1p9,v40,z100,tool0\WObj:=wobj0;
        MoveJ P1M1p10,v40,z100,tool0\WObj:=wobj0;
        MoveJ P2M1p1,v1500,z100,tool0\WObj:=wobj0;
        MoveJ P2M1p2,v40,z100,tool0\WObj:=wobj0;
        MoveJ P2M1p3,v40,z100,tool0\WObj:=wobj0;
        MoveJ P2M1p4,v40,z100,tool0\WObj:=wobj0;
        MoveJ P2M1p5,v1500,z100,tool0\WObj:=wobj0;
        MoveJ P2M1p6,v40,z100,tool0\WObj:=wobj0;
        MoveJ P2M1p7,v1500,z100,tool0\WObj:=wobj0;
        MoveJ P2M1p8,v40,z100,tool0\WObj:=wobj0;
        MoveJ P2M1p9,v40,z100,tool0\WObj:=wobj0;
        MoveJ P2M1p10,v40,z100,tool0\WObj:=wobj0;
        MoveJ P3M1p1,v1500,z100,tool0\WObj:=wobj0;
        MoveJ P3M1p2,v40,z100,tool0\WObj:=wobj0;
        MoveJ P3M1p3,v40,z100,tool0\WObj:=wobj0;
        MoveJ P3M1p4,v40,z100,tool0\WObj:=wobj0;
        MoveJ P3M1p5,v1500,z100,tool0\WObj:=wobj0;
        MoveJ P3M1p6,v40,z100,tool0\WObj:=wobj0;
        MoveJ P3M1p7,v1500,z100,tool0\WObj:=wobj0;
        MoveJ P3M1p8,v40,z100,tool0\WObj:=wobj0;
        MoveJ P3M1p9,v40,z100,tool0\WObj:=wobj0;
        MoveJ P3M1p10,v40,z100,tool0\WObj:=wobj0;
        MoveJ P4M1p1,v1500,z100,tool0\WObj:=wobj0;
        MoveJ P4M1p2,v40,z100,tool0\WObj:=wobj0;
        MoveJ P4M1p3,v40,z100,tool0\WObj:=wobj0;
        MoveJ P4M1p4,v40,z100,tool0\WObj:=wobj0;
        MoveJ P4M1p5,v1500,z100,tool0\WObj:=wobj0;
        MoveJ P4M1p6,v40,z100,tool0\WObj:=wobj0;
        MoveJ P4M1p7,v1500,z100,tool0\WObj:=wobj0;
        MoveJ P4M1p8,v40,z100,tool0\WObj:=wobj0;
        MoveJ P4M1p9,v40,z100,tool0\WObj:=wobj0;
        MoveJ P4M1p10,v40,z100,tool0\WObj:=wobj0;
        MoveJ P4M1p12,v1500,z100,tool0\WObj:=wobj0;
        MoveJ P4M1p11,v40,z100,tool0\WObj:=wobj0;
        MoveJ P3M1p12,v1500,z100,tool0\WObj:=wobj0;
        MoveJ P3M1p11,v40,z100,tool0\WObj:=wobj0;
        MoveJ P2M1p12,v1500,z100,tool0\WObj:=wobj0;
        MoveJ P2M1p11,v40,z100,tool0\WObj:=wobj0;
        MoveJ P1M1p12,v1500,z100,tool0\WObj:=wobj0;
        MoveJ P1M1p11,v40,z100,tool0\WObj:=wobj0;
        MoveJ P5M1p1,v1500,z100,tool0\WObj:=wobj0;
        MoveJ P5M1p2,v40,z100,tool0\WObj:=wobj0;
        MoveJ P5M1p3,v40,z100,tool0\WObj:=wobj0;
        MoveJ P5M1p4,v40,z100,tool0\WObj:=wobj0;
        MoveJ P5M1p5,v1500,z100,tool0\WObj:=wobj0;
        MoveJ P5M1p6,v40,z100,tool0\WObj:=wobj0;
        MoveJ P5M1p7,v1500,z100,tool0\WObj:=wobj0;
        MoveJ P5M1p8,v40,z100,tool0\WObj:=wobj0;
        MoveJ P5M1p9,v40,z100,tool0\WObj:=wobj0;
        MoveJ P5M1p10,v40,z100,tool0\WObj:=wobj0;
        MoveJ P6M1p1,v1500,z100,tool0\WObj:=wobj0;
        MoveJ P6M1p2,v40,z100,tool0\WObj:=wobj0;
        MoveJ P6M1p3,v40,z100,tool0\WObj:=wobj0;
        MoveJ P6M1p4,v40,z100,tool0\WObj:=wobj0;
        MoveJ P6M1p5,v1500,z100,tool0\WObj:=wobj0;
        MoveJ P6M1p6,v40,z100,tool0\WObj:=wobj0;
        MoveJ P6M1p7,v1500,z100,tool0\WObj:=wobj0;
        MoveJ P6M1p8,v40,z100,tool0\WObj:=wobj0;
        MoveJ P6M1p9,v40,z100,tool0\WObj:=wobj0;
        MoveJ P6M1p10,v40,z100,tool0\WObj:=wobj0;
        MoveJ P7M1p1,v1500,z100,tool0\WObj:=wobj0;
        MoveJ P7M1p2,v40,z100,tool0\WObj:=wobj0;
        MoveJ P7M1p3,v40,z100,tool0\WObj:=wobj0;
        MoveJ P7M1p4,v40,z100,tool0\WObj:=wobj0;
        MoveJ P7M1p5,v1500,z100,tool0\WObj:=wobj0;
        MoveJ P7M1p6,v40,z100,tool0\WObj:=wobj0;
        MoveJ P7M1p7,v1500,z100,tool0\WObj:=wobj0;
        MoveJ P7M1p8,v40,z100,tool0\WObj:=wobj0;
        MoveJ P7M1p9,v40,z100,tool0\WObj:=wobj0;
        MoveJ P7M1p10,v40,z100,tool0\WObj:=wobj0;
        MoveJ P8M1p1,v1500,z100,tool0\WObj:=wobj0;
        MoveJ P8M1p2,v40,z100,tool0\WObj:=wobj0;
        MoveJ P8M1p3,v40,z100,tool0\WObj:=wobj0;
        MoveJ P8M1p4,v40,z100,tool0\WObj:=wobj0;
        MoveJ P8M1p5,v1500,z100,tool0\WObj:=wobj0;
        MoveJ P8M1p6,v40,z100,tool0\WObj:=wobj0;
        MoveJ P8M1p7,v1500,z100,tool0\WObj:=wobj0;
        MoveJ P8M1p8,v40,z100,tool0\WObj:=wobj0;
        MoveJ P8M1p9,v40,z100,tool0\WObj:=wobj0;
        MoveJ P8M1p10,v40,z100,tool0\WObj:=wobj0;
        MoveJ P8M1p12,v1500,z100,tool0\WObj:=wobj0;
        MoveJ P8M1p11,v40,z100,tool0\WObj:=wobj0;
        MoveJ P7M1p12,v1500,z100,tool0\WObj:=wobj0;
        MoveJ P7M1p11,v40,z100,tool0\WObj:=wobj0;
        MoveJ P6M1p12,v1500,z100,tool0\WObj:=wobj0;
        MoveJ P6M1p11,v40,z100,tool0\WObj:=wobj0;
        MoveJ P5M1p12,v1500,z100,tool0\WObj:=wobj0;
        MoveJ P5M1p11,v40,z100,tool0\WObj:=wobj0;
        MoveJ Esperando,v1500,z100,tool0\WObj:=wobj0;
        MoveJ EsperandoMOVMesa,v1500,z100,tool0\WObj:=wobj0;
        MoveJ P1M2p1,v1500,z100,tool0\WObj:=wobj0;
        MoveJ P1M2p2,v40,z100,tool0\WObj:=wobj0;
        MoveJ P1M2p3,v40,z100,tool0\WObj:=wobj0;
        MoveJ P1M2p4,v40,z100,tool0\WObj:=wobj0;
        MoveJ P1M2p5,v1500,z100,tool0\WObj:=wobj0;
        MoveJ P1M2p6,v40,z100,tool0\WObj:=wobj0;
        MoveJ P1M2p7,v40,z100,tool0\WObj:=wobj0;
        MoveJ P1M2p8,v1500,z100,tool0\WObj:=wobj0;
        MoveJ P1M2p9,v40,z100,tool0\WObj:=wobj0;
        MoveJ P1M2p10,v40,z100,tool0\WObj:=wobj0;
        MoveJ P2M2p1,v1500,z100,tool0\WObj:=wobj0;
        MoveJ P2M2p2,v40,z100,tool0\WObj:=wobj0;
        MoveJ P2M2p3,v40,z100,tool0\WObj:=wobj0;
        MoveJ P2M2p4,v40,z100,tool0\WObj:=wobj0;
        MoveJ P2M2p5,v1500,z100,tool0\WObj:=wobj0;
        MoveJ P2M2p6,v40,z100,tool0\WObj:=wobj0;
        MoveJ P2M2p7,v40,z100,tool0\WObj:=wobj0;
        MoveJ P2M2p8,v1500,z100,tool0\WObj:=wobj0;
        MoveJ P2M2p9,v40,z100,tool0\WObj:=wobj0;
        MoveJ P2M2p10,v40,z100,tool0\WObj:=wobj0;
        MoveJ P3M2p1,v1500,z100,tool0\WObj:=wobj0;
        MoveJ P3M2p2,v40,z100,tool0\WObj:=wobj0;
        MoveJ P3M2p3,v40,z100,tool0\WObj:=wobj0;
        MoveJ P3M2p4,v40,z100,tool0\WObj:=wobj0;
        MoveJ P3M2p5,v1500,z100,tool0\WObj:=wobj0;
        MoveJ P3M2p6,v40,z100,tool0\WObj:=wobj0;
        MoveJ P3M2p7,v40,z100,tool0\WObj:=wobj0;
        MoveJ P3M2p8,v1500,z100,tool0\WObj:=wobj0;
        MoveJ P3M2p9,v40,z100,tool0\WObj:=wobj0;
        MoveJ P3M2p10,v40,z100,tool0\WObj:=wobj0;
        MoveJ P4M2p1,v1500,z100,tool0\WObj:=wobj0;
        MoveJ P4M2p2,v40,z100,tool0\WObj:=wobj0;
        MoveJ P4M2p3,v40,z100,tool0\WObj:=wobj0;
        MoveJ P4M2p4,v40,z100,tool0\WObj:=wobj0;
        MoveJ P4M2p5,v1500,z100,tool0\WObj:=wobj0;
        MoveJ P4M2p6,v40,z100,tool0\WObj:=wobj0;
        MoveJ P4M2p7,v40,z100,tool0\WObj:=wobj0;
        MoveJ P4M2p8,v1500,z100,tool0\WObj:=wobj0;
        MoveJ P4M2p9,v40,z100,tool0\WObj:=wobj0;
        MoveJ P4M2p10,v40,z100,tool0\WObj:=wobj0;
        MoveJ P4M2p12,v1500,z100,tool0\WObj:=wobj0;
        MoveJ P4M2p11,v40,z100,tool0\WObj:=wobj0;
        MoveJ P3M2p12,v1500,z100,tool0\WObj:=wobj0;
        MoveJ P3M2p11,v40,z100,tool0\WObj:=wobj0;
        MoveJ P2M2p12,v1500,z100,tool0\WObj:=wobj0;
        MoveJ P2M2p11,v40,z100,tool0\WObj:=wobj0;
        MoveJ P1M2p12,v1500,z100,tool0\WObj:=wobj0;
        MoveJ P1M2p11,v40,z100,tool0\WObj:=wobj0;
        MoveJ P5M2p1,v1500,z100,tool0\WObj:=wobj0;
        MoveJ P5M2p2,v40,z100,tool0\WObj:=wobj0;
        MoveJ P5M2p3,v40,z100,tool0\WObj:=wobj0;
        MoveJ P5M2p4,v40,z100,tool0\WObj:=wobj0;
        MoveJ P5M2p5,v1500,z100,tool0\WObj:=wobj0;
        MoveJ P5M2p6,v40,z100,tool0\WObj:=wobj0;
        MoveJ P5M2p7,v40,z100,tool0\WObj:=wobj0;
        MoveJ P5M2p8,v1500,z100,tool0\WObj:=wobj0;
        MoveJ P5M2p9,v40,z100,tool0\WObj:=wobj0;
        MoveJ P5M2p10,v40,z100,tool0\WObj:=wobj0;
        MoveJ P6M2p1,v1500,z100,tool0\WObj:=wobj0;
        MoveJ P6M2p2,v40,z100,tool0\WObj:=wobj0;
        MoveJ P6M2p3,v40,z100,tool0\WObj:=wobj0;
        MoveJ P6M2p4,v40,z100,tool0\WObj:=wobj0;
        MoveJ P6M2p5,v1500,z100,tool0\WObj:=wobj0;
        MoveJ P6M2p6,v40,z100,tool0\WObj:=wobj0;
        MoveJ P6M2p7,v40,z100,tool0\WObj:=wobj0;
        MoveJ P6M2p8,v1500,z100,tool0\WObj:=wobj0;
        MoveJ P6M2p9,v40,z100,tool0\WObj:=wobj0;
        MoveJ P6M2p10,v40,z100,tool0\WObj:=wobj0;
        MoveJ P7M2p1,v1500,z100,tool0\WObj:=wobj0;
        MoveJ P7M2p2,v40,z100,tool0\WObj:=wobj0;
        MoveJ P7M2p3,v40,z100,tool0\WObj:=wobj0;
        MoveJ P7M2p4,v40,z100,tool0\WObj:=wobj0;
        MoveJ P7M2p5,v1500,z100,tool0\WObj:=wobj0;
        MoveJ P7M2p6,v40,z100,tool0\WObj:=wobj0;
        MoveJ P7M2p7,v40,z100,tool0\WObj:=wobj0;
        MoveJ P7M2p8,v1500,z100,tool0\WObj:=wobj0;
        MoveJ P7M2p9,v40,z100,tool0\WObj:=wobj0;
        MoveJ P7M2p10,v40,z100,tool0\WObj:=wobj0;
        MoveJ P8M2p1,v1500,z100,tool0\WObj:=wobj0;
        MoveJ P8M2p2,v40,z100,tool0\WObj:=wobj0;
        MoveJ P8M2p3,v40,z100,tool0\WObj:=wobj0;
        MoveJ P8M2p4,v40,z100,tool0\WObj:=wobj0;
        MoveJ P8M2p5,v1500,z100,tool0\WObj:=wobj0;
        MoveJ P8M2p6,v40,z100,tool0\WObj:=wobj0;
        MoveJ P8M2p7,v40,z100,tool0\WObj:=wobj0;
        MoveJ P8M2p8,v1500,z100,tool0\WObj:=wobj0;
        MoveJ P8M2p9,v40,z100,tool0\WObj:=wobj0;
        MoveJ P8M2p10,v40,z100,tool0\WObj:=wobj0;
        MoveJ P8M2p12,v1500,z100,tool0\WObj:=wobj0;
        MoveJ P8M2p11,v40,z100,tool0\WObj:=wobj0;
        MoveJ P7M2p12,v1500,z100,tool0\WObj:=wobj0;
        MoveJ P7M2p11,v40,z100,tool0\WObj:=wobj0;
        MoveJ P6M2p12,v1500,z100,tool0\WObj:=wobj0;
        MoveJ P6M2p11,v40,z100,tool0\WObj:=wobj0;
        MoveJ P5M2p12,v1500,z100,tool0\WObj:=wobj0;
        MoveJ P5M2p11,v40,z100,tool0\WObj:=wobj0;
        MoveJ HomeMesaDos,v1500,z100,tool0\WObj:=wobj0;
        DeactUnit INTERCH;
    ENDPROC
ENDMODULE
